FUNCTION_BLOCK PtHelper
VAR_INPUT
END_VAR
VAR_OUTPUT
END_VAR
VAR
END_VAR

END_FUNCTION_BLOCK

(* stored: Version 1.1.0.1, ProductVersion 3.1.4024.12
   POU PtHelper: Id {9b813d75-59c2-4ce7-81be-3a81dd058dc5}, SpecialFunc None *)
